(* IEC 61131-3 sources: commands/test/ExampleCommand, 3 files *)

(* ---- ActuatorWithFeedback.st ---- *)
USING Simatic.Ax.Commands;
USING AxUnit.Assert;

NAMESPACE Simatic.Ax.Actuators

    FUNCTION_BLOCK ActuatorWithFeedback
        VAR_INPUT
            execute : BOOL;
            feedback : BOOL;
        END_VAR
        VAR_OUTPUT
            busy : BOOL;
            done : BOOL;
            error : BOOL;
            control : BOOL;
        END_VAR
        VAR
            executeOld : BOOL;
            state : INT;
        END_VAR
        VAR_TEMP
            executeRis : BOOL;
        END_VAR
        VAR CONSTANT
            STATE_IDLE : INT := 0;
            STATE_BUSY : INT := 1;
            STATE_DONE : INT := 2;
            STATE_ERROR : INT := 3;
        END_VAR

        executeRis := execute AND NOT(executeRis);
        executeOld := execute;

        CASE state OF
            STATE_IDLE:
                control := FALSE;
                busy := FALSE;
                error := FALSE;
                done := FALSE;
                IF (executeRis) THEN
                    state := STATE_BUSY;
                END_IF;
            STATE_BUSY:
            control := TRUE;
            busy := TRUE;
                IF (feedback) THEN
                    state := STATE_DONE;
                    busy := FALSE;
                    done := TRUE;
                END_IF;
            STATE_DONE:
                state := STATE_IDLE;
            STATE_ERROR: ;
        END_CASE;

    END_FUNCTION_BLOCK

END_NAMESPACE

(* ---- ControlUntilSensorHasReached.st ---- *)
USING Simatic.Ax.Commands;
USING AxUnit.Assert;

NAMESPACE Simatic.Ax.Actuators

    CLASS INTERNAL ControlUntilSensorHasReached
        EXTENDS ExecuteCommand
        VAR PUBLIC
            Feedback : REF_TO BOOL;
            Control : REF_TO BOOL;
        END_VAR
        VAR
            m_Actuator : ActuatorWithFeedback;
        END_VAR

        METHOD PUBLIC Start : itfCommand
            THIS.ExecuteWithRisingEdge();
            Start := THIS;
        END_METHOD

        METHOD PROTECTED OVERRIDE Execute
            m_Actuator(feedback := Feedback^, control => Control^, done => _done, error => _done);
        END_METHOD

        METHOD PROTECTED OVERRIDE SetExecute
            VAR_INPUT
                exec : BOOL;
            END_VAR
            m_Actuator.execute := TRUE;
            ;
        END_METHOD
    END_CLASS

END_NAMESPACE

(* ---- TwoWayActuator.st ---- *)
USING Simatic.Ax.Commands;
USING AxUnit.Assert;

NAMESPACE Simatic.Ax.Actuators
    CLASS TwoWayActuator
        VAR PUBLIC
            controlToWorkPos : BOOL;
            feedbackInWorkPos : BOOL;
            controlToHomePos : BOOL;
            feedbackInHomePos: BOOL;
        END_VAR
        VAR PROTECTED
            _toHomePos : ControlUntilSensorHasReached;
            _toWorkPos : ControlUntilSensorHasReached;
        END_VAR

        METHOD PUBLIC Init
            _toWorkPos.Control := REF(controlToWorkPos);
            _toWorkPos.Feedback := REF(feedbackInWorkPos);
            _toHomePos.Control := REF(controlToHomePos);
            _toHomePos.Feedback := REF(feedbackInHomePos);
        END_METHOD

        METHOD PUBLIC GoToWorkPos : itfCommand
            GoToWorkPos := _toWorkPos.Start();
        END_METHOD

        METHOD PUBLIC GoToHomePos : itfCommand
            GoToHomePos := _toHomePos.Start();
        END_METHOD

    END_CLASS
END_NAMESPACE
